TYPE ST_ProcessingDatasets :
    STRUCT
    lrColFirstRowRedundancy    : LREAL := 10; // 首行提前量%


lrColRowOverlap          : LREAL := 0; // 前后行重叠量%


lrRowStartPositionDis    : LREAL := 40.000; // 行开始位置与中心点间距


lrRowInVeloPositionDis   : LREAL := 30.000; // 行到达匀速点与中心点间距


lrRowTriggerTakePhotoDis : LREAL := 10.000;
    lrRowTriggerStopPhotoDis   : LREAL := 10.000;
    lrRowEndConstantSpdDis     : LREAL := 25.000;
    lrRowStopMoveDis           : LREAL := 30.000;
    END_STRUCT
END_TYPE

(* stored: Version 1.1.0.1, ProductVersion 3.1.4024.12
   DUT ST_ProcessingDatasets: Id {ab9b9c4a-2ccc-4b43-8ff8-569b8c5273cf} *)
